Staubli VAL3: pp_cell_bk.pgx

program pp_cell_bk()
  local num l_nNum_f2_lim
  local num l_nNum_f3_lim
  local num l_nNum_f2_idx
  local num l_nNum_f3_idx
  local num l_nNum_cRow
  local num l_nNum_cCol
  local point l_pPoint_cur
begin
  //---------------------------------
  //from cells(f2,f3) to back secure
  //---------------------------------

   //initialize
  call calculate_total(2,l_nNum_f2_lim)
  call calculate_total(3,l_nNum_f3_lim)

  l_nNum_f2_idx = 0
  l_nNum_f3_idx = 0

  while true

    //reload  reminder
    call show_check("Recycle pp_cell_bk")

    //----------
    //f2 cell pick
    //------------

    //runout remider
    if l_nNum_f2_idx >= l_nNum_f2_lim
      //warning if runs out
      call show_check("Reload F2")
      //reset
      l_nNum_f2_idx = 0
    endIf

    call calculate_rc(l_nNum_f2_idx,2,l_nNum_cRow,l_nNum_cCol)
    call calculate_pick(l_nNum_cRow,l_nNum_cCol,l_pPoint_cur,2)
    call regular_pick(t2,mNomSpeed,mSlowSpeed,l_pPoint_cur,dDio_t2_cy,false,dDio_f2_secure)
    //show progress
    call show_progress(sScreen_ppShelf,l_nNum_f2_idx+1,l_nNum_f2_lim,7)
    //increase
    l_nNum_f2_idx = l_nNum_f2_idx +1

    //-------
    //f3pick
    //-------

    //runout reminder
    if l_nNum_f3_idx >= l_nNum_f3_lim
      //warning if runs out
      call show_check("Reload F3")
      //reset
      l_nNum_f3_idx = 0
    endIf
    call calculate_rc(l_nNum_f3_idx,3,l_nNum_cRow,l_nNum_cCol)
    call calculate_pick(l_nNum_cRow,l_nNum_cCol,l_pPoint_cur,3)
    call regular_pick(t3,mNomSpeed,mSlowSpeed,l_pPoint_cur,dDio_t3_cy,false,dDio_f3_secure)
    //show progress
    call show_progress(sScreen_ppShelf,l_nNum_f3_idx+1,l_nNum_f3_lim,8)
    //increase
    l_nNum_f3_idx = l_nNum_f3_idx +1

    //--------------
    //pp back secure
    //--------------
    call pp_back_secure()

    //-------------
    // drop
    //-------------
    call regular_place(t3,mNomSpeed,mSlowSpeed,pPointRx_f3_bk,false,dDio_t3_cy,false)


  endWhile


end
